FUNCTION_BLOCK FB_SITP_SygnalizacjaStanu_Resetting EXTENDS FB_SITP_SygnalizacjaStanu
VAR
END_VAR

METHOD PUBLIC UstawPrace
VAR_INPUT
END_VAR

THIS^.refarrLampki [E_SITP_LampkiSygnalizacyjne.WiezaCzerwona].Wlacz2		(bSwiec := TRUE, 	bMigaj := FALSE,	 tWlaczony := T#0MS,	 tWylaczony := T#0MS);(*			Czerwona		*)
THIS^.refarrLampki [E_SITP_LampkiSygnalizacyjne.WiezaZolta].Wlacz2			(bSwiec := FALSE, 	bMigaj := FALSE,	 tWlaczony := T#0MS,	 tWylaczony := T#0MS);(*			Zółta			*)
THIS^.refarrLampki [E_SITP_LampkiSygnalizacyjne.WiezaZielona].Wlacz2		(bSwiec := TRUE, 	bMigaj := FALSE,	 tWlaczony := T#0MS,	 tWylaczony := T#0MS);(*			Zielona			*)
THIS^.refarrLampki [E_SITP_LampkiSygnalizacyjne.WiezaBiala].Wlacz2			(bSwiec := FALSE, 	bMigaj := FALSE,	 tWlaczony := T#0MS,	 tWylaczony := T#0MS);(*			Niebieska		*)
THIS^.refarrLampki [E_SITP_LampkiSygnalizacyjne.WiezaNiebieska].Wlacz2		(bSwiec := FALSE, 	bMigaj := FALSE,	 tWlaczony := T#0MS,	 tWylaczony := T#0MS);(*			Biała			*)



THIS^.refarrLampki [E_SITP_LampkiSygnalizacyjne.PrzyciskStart].Wlacz2		(bSwiec := TRUE, 	bMigaj := FALSE,	 tWlaczony := T#0MS,	 tWylaczony := T#0MS);(*	Lampka przycisku Start    	*)
THIS^.refarrLampki [E_SITP_LampkiSygnalizacyjne.PrzyciskStop].Wlacz2		(bSwiec := TRUE, 	bMigaj := FALSE,	 tWlaczony := T#0MS,	 tWylaczony := T#0MS);(*	Lampka przycisku Stop     	*)
THIS^.refarrLampki [E_SITP_LampkiSygnalizacyjne.PrzyciskHold].Wlacz2		(bSwiec := FALSE, 	bMigaj := FALSE,	 tWlaczony := T#0MS,	 tWylaczony := T#0MS);(*	Lampka przycisku Hold     	*)
THIS^.refarrLampki [E_SITP_LampkiSygnalizacyjne.PrzyciskUnhold].Wlacz2		(bSwiec := FALSE, 	bMigaj := FALSE,	 tWlaczony := T#0MS,	 tWylaczony := T#0MS);(*	Lampka przycisku Unhold   	*)
THIS^.refarrLampki [E_SITP_LampkiSygnalizacyjne.PrzyciskSuspend].Wlacz2		(bSwiec := FALSE, 	bMigaj := FALSE,	 tWlaczony := T#0MS,	 tWylaczony := T#0MS);(*	Lampka przycisku Suspend  	*)
THIS^.refarrLampki [E_SITP_LampkiSygnalizacyjne.PrzyciskUnsuspend].Wlacz2	(bSwiec := FALSE, 	bMigaj := FALSE,	 tWlaczony := T#0MS,	 tWylaczony := T#0MS);(*	Lampka przycisku Unsuspend	*)
THIS^.refarrLampki [E_SITP_LampkiSygnalizacyjne.PrzyciskAbort].Wlacz2		(bSwiec := FALSE, 	bMigaj := FALSE,	 tWlaczony := T#0MS,	 tWylaczony := T#0MS);(*	Lampka przycisku Abort    	*)
THIS^.refarrLampki [E_SITP_LampkiSygnalizacyjne.PrzyciskClear].Wlacz2		(bSwiec := FALSE, 	bMigaj := FALSE,	 tWlaczony := T#0MS,	 tWylaczony := T#0MS);(*	Lampka przycisku Clear    	*)
THIS^.refarrLampki [E_SITP_LampkiSygnalizacyjne.PrzyciskComplete].Wlacz2	(bSwiec := FALSE, 	bMigaj := FALSE,	 tWlaczony := T#0MS,	 tWylaczony := T#0MS);(*	Lampka przycisku Complete	*)
END_METHOD

END_FUNCTION_BLOCK

(* stored: Version 1.1.0.1
   POU FB_SITP_SygnalizacjaStanu_Resetting: Id {6f636098-1ab8-0075-2330-aaf2db942b74}, SpecialFunc None
   Method UstawPrace: Id {e5214150-9ae1-0f2a-21fc-e203a6f9f77c} *)
